// Mitsubishi GX Works2 project: counter2   PLC: Q03UDV

PROGRAM MAIN
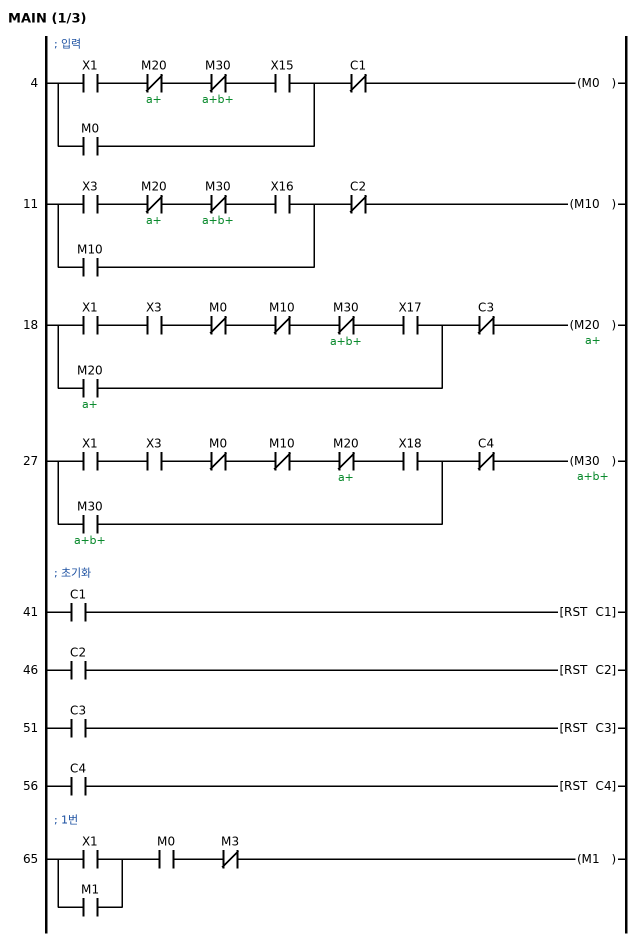
; 입력
4     LD      X1
      ANI     M20  ; a+
      ANI     M30  ; a+b+
      AND     X15
      OR      M0
      ANI     C1
      OUT     M0
11    LD      X3
      ANI     M20  ; a+
      ANI     M30  ; a+b+
      AND     X16
      OR      M10
      ANI     C2
      OUT     M10
18    LD      X1
      AND     X3
      ANI     M0
      ANI     M10
      ANI     M30  ; a+b+
      AND     X17
      OR      M20  ; a+
      ANI     C3
      OUT     M20  ; a+
27    LD      X1
      AND     X3
      ANI     M0
      ANI     M10
      ANI     M20  ; a+
      AND     X18
      OR      M30  ; a+b+
      ANI     C4
      OUT     M30  ; a+b+
; 초기화
41    LD      C1
      RST     C1
46    LD      C2
      RST     C2
51    LD      C3
      RST     C3
56    LD      C4
      RST     C4
; 1번
65    LD      X1
      OR      M1
      AND     M0
      ANI     M3
      OUT     M1
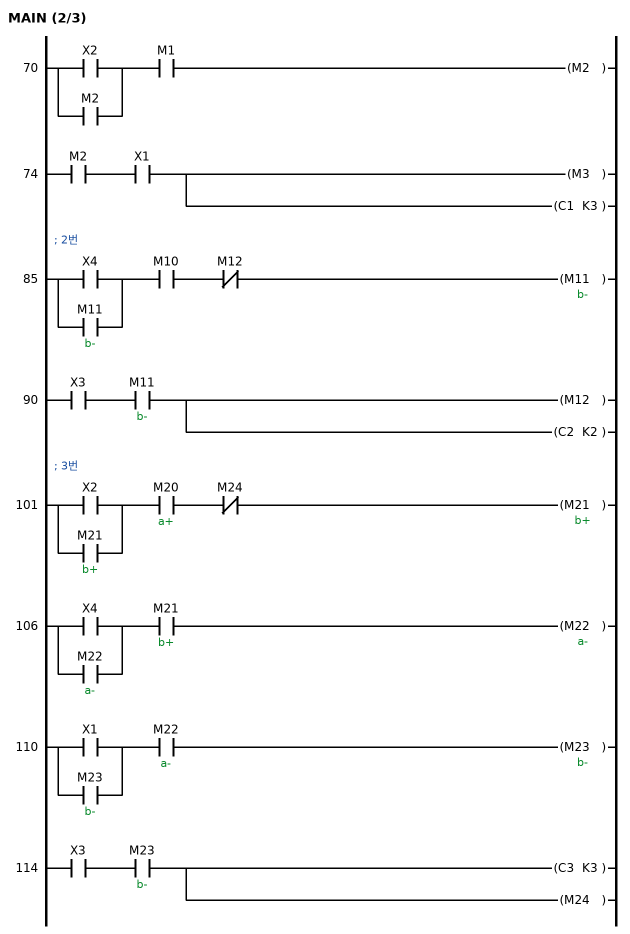
70    LD      X2
      OR      M2
      AND     M1
      OUT     M2
74    LD      M2
      AND     X1
      OUT     M3
      OUT     C1 K3
; 2번
85    LD      X4
      OR      M11  ; b-
      AND     M10
      ANI     M12
      OUT     M11  ; b-
90    LD      X3
      AND     M11  ; b-
      OUT     M12
      OUT     C2 K2
; 3번
101   LD      X2
      OR      M21  ; b+
      AND     M20  ; a+
      ANI     M24
      OUT     M21  ; b+
106   LD      X4
      OR      M22  ; a-
      AND     M21  ; b+
      OUT     M22  ; a-
110   LD      X1
      OR      M23  ; b-
      AND     M22  ; a-
      OUT     M23  ; b-
114   LD      X3
      AND     M23  ; b-
      OUT     C3 K3
      OUT     M24
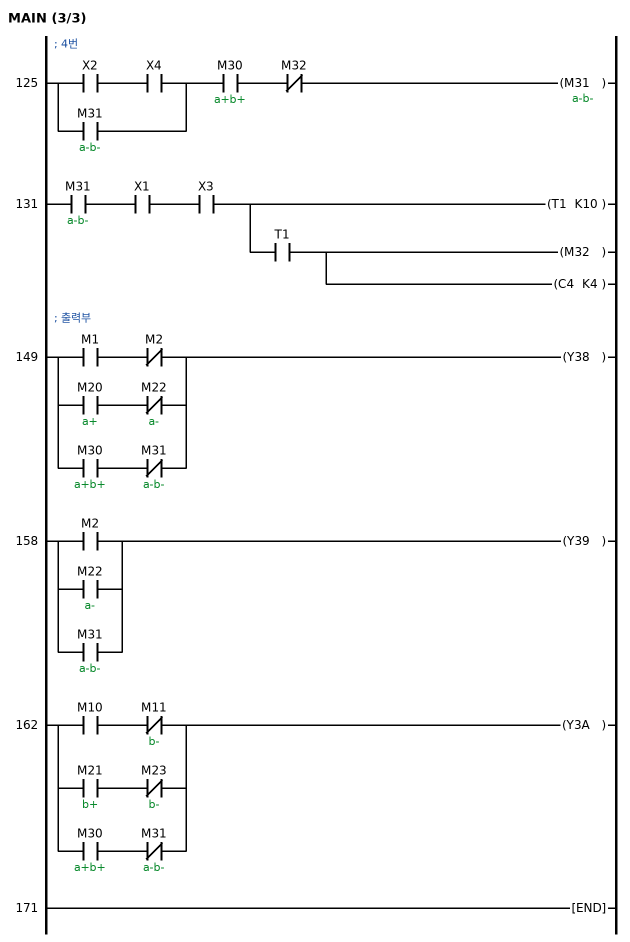
; 4번
125   LD      X2
      AND     X4
      OR      M31  ; a-b-
      AND     M30  ; a+b+
      ANI     M32
      OUT     M31  ; a-b-
131   LD      M31  ; a-b-
      AND     X1
      AND     X3
      OUT     T1 K10
      AND     T1
      OUT     M32
      OUT     C4 K4
; 출력부
149   LD      M1
      ANI     M2
      LD      M20  ; a+
      ANI     M22  ; a-
      ORB
      LD      M30  ; a+b+
      ANI     M31  ; a-b-
      ORB
      OUT     Y38
158   LD      M2
      OR      M22  ; a-
      OR      M31  ; a-b-
      OUT     Y39
162   LD      M10
      ANI     M11  ; b-
      LD      M21  ; b+
      ANI     M23  ; b-
      ORB
      LD      M30  ; a+b+
      ANI     M31  ; a-b-
      ORB
      OUT     Y3A
171   END
END_PROGRAM
